Fanuc KAREL source: GET_TPE_PRM.kl

PROGRAM T
%NOLOCKGROUP
VAR
 v0 : INTEGER
 v1 : INTEGER
 v2 : INTEGER
 v3 : REAL
 v4 : STRING[40]
 v5 : INTEGER
BEGIN
 GET_TPE_PRM(v0, v1, v2, v3, v4, v5)
END T
